PROGRAM FillBox
VAR
		BoxCylinder				:	BOOL; 	// cylinder to stop box to be filled
		ItemReady				:	BOOL;	// item ready to be moved to the box by the robot
		StartRobotPrg			:	BOOL;	// start robot program
		RobotMoveOneItem		:	BOOL;	// signal to robot: move one item
		BoxReadyToFill			:	BOOL;	// a box is ready to be filled
		RobotMovedAllItems		: 	BOOL;	// signal from robot. Robot has moved all items
END_VAR
VAR // added by the converter: edge detectors and wires of the graphical bodies
    _w1 : BOOL;
END_VAR

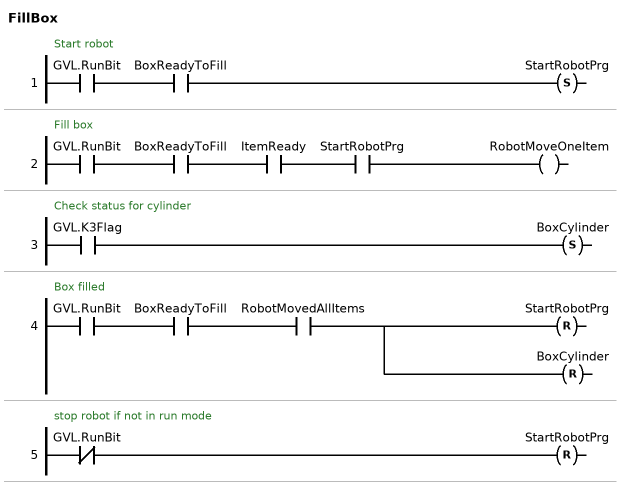
// NETWORK 1
// Start robot
StartRobotPrg S= GVL.RunBit AND BoxReadyToFill;

// NETWORK 2
// Fill box
RobotMoveOneItem := GVL.RunBit AND BoxReadyToFill AND ItemReady AND StartRobotPrg;

// NETWORK 3
// Check status for cylinder
BoxCylinder S= GVL.K3Flag;

// NETWORK 4
// Box filled
_w1 := GVL.RunBit AND BoxReadyToFill AND RobotMovedAllItems;
StartRobotPrg R= _w1;
BoxCylinder R= _w1;

// NETWORK 5
// stop robot if not in run mode
StartRobotPrg R= NOT GVL.RunBit;

END_PROGRAM

(* stored: Version 1.1.0.1, ProductVersion 3.1.4024.15
   POU FillBox: Id {5ca92c9d-f67a-443f-9d7e-ab3c76bd689e}, SpecialFunc None *)
